{attribute 'qualified_only'}
VAR_GLOBAL
	sNetId				: T_AmsNetId := '5.109.65.175.2.1';
	nSlaveAddr			: UINT := 1004;
	
	Controlword AT%Q*		: UINT;	
	Statusword AT%I*		: UINT;
	
	bReset					: BOOL;
END_VAR

(* stored: Version 1.1.0.1, ProductVersion 3.1.4024.11
   GVL GVL: Id {03894085-25e2-4207-96ab-602d7bd3dadd} *)
